(* PLC project Blank Project, Blank Blank 1.0 *)
(* stored: creationDateTime 2016-05-18T21:14:07, modificationDateTime 2016-11-21T18:24:04 *)

PROGRAM Cell2
  VAR
    C1_IR AT %IX0.3 : BOOL := true;
    M1_IR AT %IX0.4 : BOOL := true;
    Main AT %IX0.6 : BOOL := true;
    M1_motor AT %QX0.2 : BOOL := true;
    C2_motor AT %QX0.4 : BOOL := true;
  END_VAR
  VAR
    C2_working : BOOL := false;
  END_VAR
  VAR
    C2_working_int AT %MD1 : DINT := 0;
  END_VAR
  VAR
    M1_working : BOOL := false;
  END_VAR
  VAR
    M1_working_int AT %MD3 : DINT := 0;
  END_VAR
  VAR
    Timer_conveyor : TON;
    Timer_machining : TON;
  END_VAR

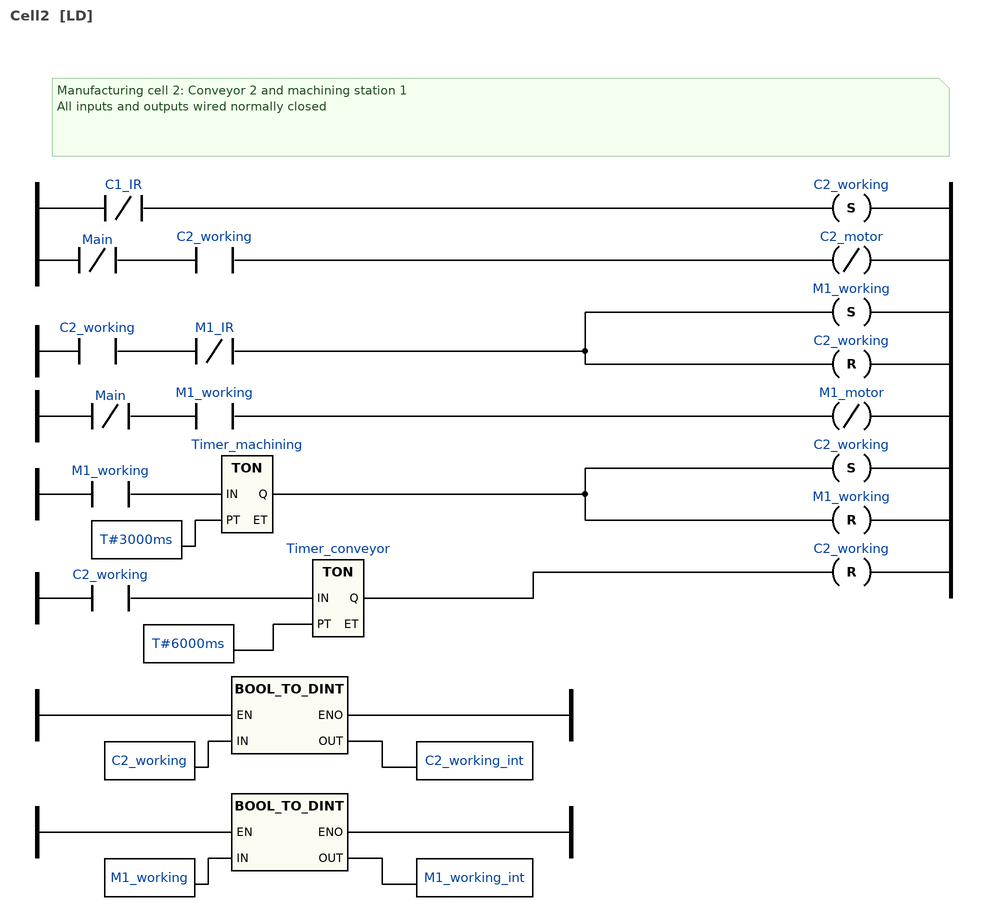
(* LD diagram, written out as Structured Text *)
(* Manufacturing cell 2: Conveyor 2 and machining station 1
All inputs and outputs wired normally closed *)
IF NOT C1_IR THEN C2_working := TRUE; END_IF;
C2_motor := NOT (NOT Main AND C2_working);
IF C2_working AND NOT M1_IR THEN M1_working := TRUE; END_IF;
IF C2_working AND NOT M1_IR THEN C2_working := FALSE; END_IF;
M1_motor := NOT (NOT Main AND M1_working);
Timer_machining(IN := M1_working, PT := T#3000ms);
IF Timer_machining.Q THEN C2_working := TRUE; END_IF;
IF Timer_machining.Q THEN M1_working := FALSE; END_IF;
Timer_conveyor(IN := C2_working, PT := T#6000ms);
IF Timer_conveyor.Q THEN C2_working := FALSE; END_IF;
C2_working_int := BOOL_TO_DINT(C2_working);
M1_working_int := BOOL_TO_DINT(M1_working);
END_PROGRAM

CONFIGURATION Config0
  RESOURCE Res0 ON PLC
    TASK TaskMain(INTERVAL := T#50ms, PRIORITY := 0);
    PROGRAM Inst0 WITH TaskMain : Cell2;
  END_RESOURCE
END_CONFIGURATION
